FUNCTION_BLOCK AX_E_PERMIT_1 (* Permissive propagation of 1 event channel with adapter (generic FB) *)
  (* Standard: 61499-1 Annex A; Description: Copyright (c) 2026 Meisterschulen am Ostbahnhof This program and the accompanying materials are made available under the terms of the Eclipse Public License 2.0 which is available at https://www.eclipse.org/legal/epl-2.0/ SPDX-License-Identifier: EPL-2.0 *)
  (* Version 1.0, 2026-09-10, Franz Höpfinger, Meisterschulen am Ostbahnhof, initial implementation *)
  PACKAGE adapter::events::unidirectional;
  {SET_ATTRIBUTE(eclipse4diac::core::GenericClassName, 'GEN_AX_E_PERMIT')}
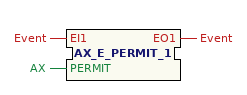
  EVENT_INPUT
    EI1; (* Event input channel 1 *)
  END_EVENT
  EVENT_OUTPUT
    EO1; (* Event output channel 1 *)
  END_EVENT
  SOCKETS
    PERMIT : adapter::types::unidirectional::AX; (* Permit condition adapter input *)
  END_SOCKETS
END_FUNCTION_BLOCK
